INTERFACE IValve

PROPERTY Value : LREAL
GET
END_GET
END_PROPERTY

END_INTERFACE

(* stored: Version 1.1.0.1, ProductVersion 3.1.4026.6
   Itf IValve: Id {c418efc0-7fa7-477a-b160-97b4e66d5689}
   Property Value: Id {39aaeb44-5b34-4f55-a98d-bb5658807dc4}
   Get Get: Id {8f450a79-a271-4dc4-a003-db3696f7e2df} *)
